TYPE AxisFeedback :
STRUCT
	Status			: BOOL;
	Busy			: BOOL;
	Active			: BOOL;
	Error			: BOOL;
	ErrorID			: UDINT;	
	Done			: BOOL;
	CommandAborted	: BOOL;
END_STRUCT
END_TYPE

(* stored: Version 1.1.0.1, ProductVersion 3.1.4024.10
   DUT AxisFeedback: Id {e9686ea9-dc3e-4cef-abb3-de4ec4310fae} *)
